FUNCTION_BLOCK OUT_COLOR (* COLOR Output *)
  (* Standard: 61499-1; Classification: HMI; Function: COLOR output *)
  (* Version 0.1, 2002-05-03, JHC, Rockwell Automation, Made QI IV=true. *)
  (* Version 0.0, 2001-04-14, JHC, Rockwell Automation, First XML version. *)
  (* Compiler header: package fb.rt.hmi; import java.awt.*; *)
  (* Compiler Java IBM VisualAge 3.0 *)
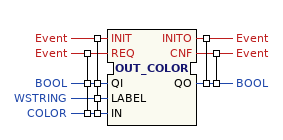
  EVENT_INPUT
    INIT WITH QI, LABEL, IN; (* Initialization *)
    REQ WITH QI, IN; (* Request *)
  END_EVENT
  EVENT_OUTPUT
    INITO WITH QO; (* Initialization Confirm *)
    CNF WITH QO; (* Service Confirmation *)
  END_EVENT
  VAR_INPUT
    QI : BOOL := true; (* Input event qualifier *)
    LABEL : WSTRING; (* Output label *)
    IN : COLOR; (* Output value *)
  END_VAR
  VAR_OUTPUT
    QO : BOOL; (* Output event qualifier *)
  END_VAR
  SERVICE OUT_COLOR/Canvas
    SEQUENCE normal_initialization
      OUT_COLOR.INIT+(DIA,IN) -> Canvas.drawOval() -> OUT_COLOR.INITO+();
    END_SEQUENCE
    SEQUENCE initialization_inhibited
      OUT_COLOR.INIT-() -> OUT_COLOR.INITO-();
    END_SEQUENCE
    SEQUENCE normal_data_transfer
      OUT_COLOR.REQ+(IN) -> Canvas.drawOval(IN) -> OUT_COLOR.CNF+();
    END_SEQUENCE
    SEQUENCE upstream_error
      OUT_COLOR.REQ-() -> OUT_COLOR.CNF-();
    END_SEQUENCE
  END_SERVICE
END_FUNCTION_BLOCK
